// TIA Portal V16 export
// export: Created 2020-03-18T18:56:42.176653Z, ExportSetting None, DisplayName Totally Integrated Automation Portal, DisplayVersion V16, DisplayName TIA Portal Version Control Interface, DisplayVersion V16, DisplayName TIA Portal Openness, DisplayVersion V16, DisplayName STEP 7 Professional, DisplayVersion V16, DisplayName STEP 7 Safety, DisplayVersion V16, DisplayName WinCC Advanced, DisplayVersion V16
FUNCTION_BLOCK "FB_EMPTY_ADAPTER"   // FB461, SCL
{ S7_Optimized_Access := 'TRUE' }
// stored: AutoNumber false, MemoryReserve 100, SetENOAutomatically false
   VAR_INPUT
      I_Start : Bool;   // Start manuell // start manual
      I_ReleaseStart : Bool;   // Freigabe start // release start
      I_ReqAbort : Bool;   // Anforderung Abbruch // request abort
      I_WaitTimeRelieve : Time;   // Wartezeit Entlasten // Waiting time relieve
      I_WaitTimeEmptying : Time;   // Wartezeit Entleeren // Waiting Time emptying
   END_VAR
   VAR_OUTPUT
      O_InitalState : Bool;   // Grundstellung // inital state
      O_Relieve : Bool;   // Entlasten // relieve
      O_Emptying : Bool;   // Entleeren // emptying
      O_WaitForOperator : Bool;   // Warten auf Benutzer // wait for operator
      O_EmptyingActive : Bool;   // Entleeren aktiv // emptying active
      O_ActualStep : Int;   // Aktueller Schritt // actual step
   END_VAR
   VAR
      ActualStep : Int;   // Aktueller Schritt // actual step
      WaitTimeRelieve { S7_SetPoint := 'True'} : TON_TIME;   // Wartezeit Entlasten // Waiting time relieve
      WaitTimeEmptying { S7_SetPoint := 'True'} : TON_TIME;   // Wartezeit Entleeren // waiting time emptying
   END_VAR
   VAR_TEMP
      Tmp_WaitTimeRelieve : Bool;   // Wartezeit Entlasten // Waiting time relieve
      Tmp_WaitTimeEmptying : Bool;   // Wartezeit Entleeren// waiting time emptying
   END_VAR
BEGIN
   // +++++++++++++++++++++++++++++++++++++++++++++++++++++++++++++++++++++++++++++++++
   // FB x460 SAT Standard Baustein // SAT standard function block
   // Erstellt / created: 03.01.2018 CSS  
   // Version / version: 0.1
   // Geändert modification: 
   // 
   // Funktion:
   // Der Baustein steuert das Entleeren eines Adapters/Füllschlauchs.
   // 
   // Function:
   // This function block controls the emptying of a adapter/hose
   // By the input config the function block switches between the brake / cooler
   // and scr mode.
   // ++++++++++++++++++++++++++++++++++++++++++++++++++++++++++++++++++++++++++++++++++ 
   // ----------------------------------------------------------------------------------
   // Zustände // states:
   // 0: Grundstellung // inital state
   // 1: Entlasten // relieve
   // 2: Schlauch/Adapter entleeren // emptying hose/adapter 
   // 3: Warten auf Benutzer // wait for operator 
   // ----------------------------------------------------------------------------------
   // 
   // Wartezeiten // waiting time
   #WaitTimeRelieve(IN := #ActualStep = 1,
                        PT := #I_WaitTimeRelieve,
                        Q => #Tmp_WaitTimeRelieve);

   #WaitTimeEmptying(IN := #ActualStep = 2 ,
                     PT := #I_WaitTimeEmptying,
                     Q => #Tmp_WaitTimeEmptying);
   // 
   // Schritte // steps
   CASE #ActualStep OF
       0: // Grundstellung // inital state
           IF (#I_ReleaseStart AND #I_Start) THEN
               #ActualStep := 1;
           END_IF;
       1: // Entlasten // relieve
           IF (#I_ReqAbort = false AND #Tmp_WaitTimeRelieve) THEN
               #ActualStep := 2;
           ELSIF #I_ReqAbort = true THEN
               #ActualStep := 0;
           END_IF;
       2: // Entleeren // emptying
           IF (#I_ReqAbort = false AND #Tmp_WaitTimeEmptying) THEN
               #ActualStep := 3;
           ELSIF #I_ReqAbort = true THEN
               #ActualStep := 0;
           END_IF;
       3: // Warten auf Benutzer // wait for operator 
           IF (#I_ReqAbort = TRUE) THEN
               #ActualStep := 0;
           END_IF;
   END_CASE;

   // Ausgabe Schritte // Output step information 
   #O_ActualStep := #ActualStep;
   #O_EmptyingActive := (#ActualStep > 0);
   // 
   #O_InitalState := (#ActualStep = 0);
   #O_Relieve := (#ActualStep = 1);
   #O_Emptying := (#ActualStep = 2);
   #O_WaitForOperator := (#ActualStep = 3);
END_FUNCTION_BLOCK
